FUNCTION_BLOCK FB_StringBuilder IMPLEMENTS I_StringBuilder
VAR
	sContent : STRING; // Store temporary strings;
END_VAR

METHOD Append : I_StringBuilder
VAR_INPUT
	sText : STRING;
END_VAR
sContent := CONCAT(STR1 := sContent, STR2 := sText);
Append := THIS^;
END_METHOD

METHOD Clear : I_StringBuilder
VAR_INPUT
END_VAR
sContent := '';
Clear := THIS^;
END_METHOD

METHOD ToString : STRING
VAR_INPUT
END_VAR
ToString := sContent; // return internal content
END_METHOD

END_FUNCTION_BLOCK

(* stored: Version 1.1.0.1, ProductVersion 3.1.4024.12
   POU FB_StringBuilder: Id {98bc1338-5d0e-4cea-931a-5879a9d2129d}, SpecialFunc None
   Method Append: Id {ee09be03-3800-4e07-8f32-47f814982d7b}
   Method Clear: Id {e057b2ee-371b-4210-9f1d-bdbe24a2ed4d}
   Method ToString: Id {96acf144-c8a6-4d52-bd4f-1b55bad3867a} *)
